Universal Robots PolyScope program: sandFront.urp

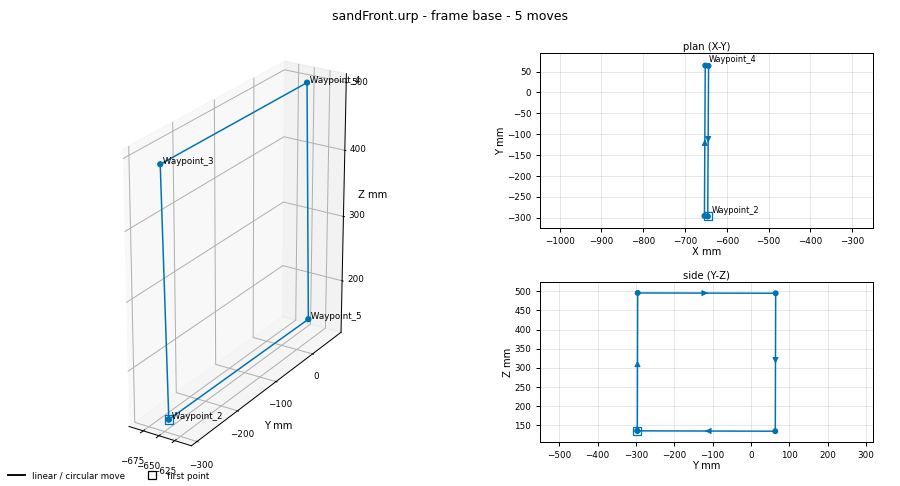
[picture p0: tool path of sandFront.urp in frame base, 5 of 5 moves have a stored position in this frame; points joined in program order, loops and branches not executed]
Program sandFront (installation=April22Cube directory=/programs/April2022Sand/subs createdIn=5.11.5.1010327 lastSavedIn=5.11.5.1010327 robotSerialNumber=20215500677)
Calibrated DH parameters: a=[0.000204, -0.239222, -0.391845, -0.000001, 0.000022, 0]; d=[0.162722, -355.808559, 353.37206, 2.570385, 0.099741, 0.099629]; alpha=[1.571124, 0.000988, 0.008295, 1.568963, -1.570303, 0]; deltaTheta=[0, -0.973091, 7.204745, 0.05153, 0, 0]
Robot Program (runOnlyOnce=true)
  Folder sandFront
    Set NoAction tcp=SandTCP
    MoveL speed 250 mm/s, acceleration 1200 mm/s^2 (useActiveTCP=false) tcp=SandTCP; feature=CubeFront
      Waypoint Waypoint_2: TCP in base x=-645.398 y=-296.455 z=135.894 mm, rx=-1.2299 ry=-1.2203 rz=1.1965 rad; joints [20.532, -26.698, 86.988, 74.06, -105.434, -14.586] deg; TCP offset x=3.18 y=114.64 z=98.2 mm, rx=-0.7854 ry=0 rz=0 rad; feature pose in base x=-150.564 y=-110.257 z=792.369 mm, rx=-0.0207 ry=-0.0133 rz=3.0697 rad
      URCap Zero FT Sensor (Robotiq_Copilot, Robotiq Inc.) dataModel(NodeInitializedKey=true, WaitForSteadyWrenchOptionKey=true, HackTriggeringContributionIsDefinedMethodKey=true)
      MoveDirectionNode (selectedDirection=ZPlus toolParams=0.05, 1.2) feature=Joint_6_name
        Until TOOL_CONTACT_DETECTION (allowActions=false retraction=NONE decelerationAcceleration=3 decelerationAngularAcceleration=34.906585)
      URCap Finishing Tool Control (Robotiq_Copilot, Robotiq Inc.) dataModel(ToolOutputNameKey=SanderOn, HackTriggeringContributionIsDefinedMethodKey=true)
      Wait Sleep waitTime=1
    MoveL speed 120 mm/s, acceleration 1200 mm/s^2 (useActiveTCP=false) tcp=SandTCP; feature=CubeFront
      URCap Zero FT Sensor (Robotiq_Copilot, Robotiq Inc.) dataModel(NodeInitializedKey=true, WaitForSteadyWrenchOptionKey=false, HackTriggeringContributionIsDefinedMethodKey=true)
      Force Simple feature=Joint_6_name; selection=[0, 0, 1, 0, 0, 0]; wrench=[0, 0, 1, 0, 0, 0]; limitsForce=[0.15, 0.15, 0.15, 1.047198, 1.047198, 1.047198]; limitsMotion=[0.1, 0.1, 0.1, 0.349066, 0.349066, 0.349066]
        Waypoint Waypoint_3: TCP in base x=-653.335 y=-295.509 z=495.795 mm, rx=-1.2297 ry=-1.2204 rz=1.1965 rad; joints [20.051, -59.037, 82.186, 111.364, -105.042, -13.942] deg
        Waypoint Waypoint_4: TCP in base x=-651.379 y=64.515 z=494.966 mm, rx=-1.2297 ry=-1.2202 rz=1.1965 rad; joints [-25.966, -70.491, 99.418, 104.332, -72.274, 18.732] deg
        Waypoint Waypoint_5: TCP in base x=-643.444 y=63.548 z=135.045 mm, rx=-1.2296 ry=-1.2202 rz=1.1965 rad; joints [-26.244, -31.945, 104.603, 60.633, -72.073, 18.608] deg
        Waypoint Waypoint_6: TCP in base x=-645.385 y=-296.43 z=135.968 mm, rx=-1.2296 ry=-1.2201 rz=1.1966 rad; joints [20.529, -26.7, 86.987, 74.045, -105.424, -14.592] deg
        URCap Finishing Tool Control (Robotiq_Copilot, Robotiq Inc.) dataModel(ToolOutputNameKey=SanderOn, FinishingToolStateKey=false, HackTriggeringContributionIsDefinedMethodKey=true)
      MoveDirectionNode (selectedDirection=ZMinus) feature=Joint_6_name
        Until DISTANCE (allowActions=false deceleration=3 distanceNodeType=STOP) Distance=0.025; motionParameters(blendRadius=0)
